PROGRAM MAIN
VAR
	fbrtmode : FB_RtMode; 
	n :DINT; 
END_VAR

n := n+1; 
//Using ADS
MAIN_ExternalTick(); 
MAIN_FastAsPossible();
 
//Using ITc
MAIN_ExternalTick_ITc(); 
MAIN_FastAsPossible_ITc(); 

//Using Functions 
MAIN_ExternalTick_F(); 
MAIN_SelfTicks_F(); 
MAIN_FastAsPossible_F();

END_PROGRAM

(* stored: Version 1.1.0.1, ProductVersion 3.1.4026.3
   POU MAIN: Id {6d192366-32dc-4bff-a587-2db1831cc73a}, SpecialFunc None *)
